FUNCTION_BLOCK Enviorment
VAR_INPUT
END_VAR
VAR_OUTPUT
END_VAR
VAR
END_VAR

METHOD Boundry 
VAR_INPUT
END_VAR
END_METHOD

METHOD Forces 
VAR_INPUT
END_VAR
END_METHOD

END_FUNCTION_BLOCK

(* stored: Version 1.1.0.1, ProductVersion 3.1.4024.12
   POU Enviorment: Id {bc804a70-ba27-434f-a722-0a692fdcb6d7}, SpecialFunc None
   Method Boundry: Id {bdc5a1ba-4bdc-4f6e-891d-211745460f60}
   Method Forces: Id {97bf2863-1c46-48a8-8c41-067ed868cafd} *)
